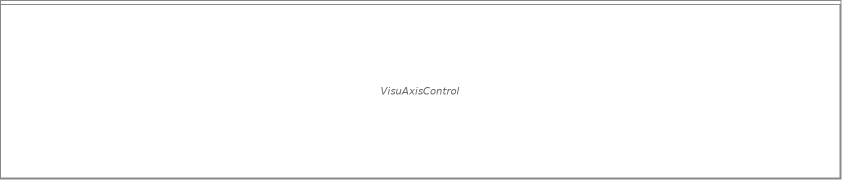
VISUALIZATION VisuAxisM2  // 842x180
    Frame (0,4 840x174)
        shows VisuAxisControl(sAxisName := sAxisM2_CName, stAxisVisu := stAxisM2_C)
END_VISUALIZATION

(* stored: Version 1.1.0.1, ProductVersion 3.1.4022.6
   Visu VisuAxisM2: Id {24c15d77-dab7-4d9d-b81e-8105768f1881} *)
